(* IEC 61131-3 sources: Industry-PLC-LLM/data/PLCBEAD_repo/PLCBEAD_PLCEmbed-main/PLC-BEAD/Source/GEB/TEMP_SI, 1 file *)

(* ---- TEMP_SI.ST ---- *)
FUNCTION TEMP_SI:REAL
	VAR_INPUT
		RES :	REAL;
		VAR_RS:	REAL;
		TS :	REAL;
	END_VAR

	TEMP_SI := (-7.64E-3 + SQRT(RES/VAR_RS* 6.64E-5 - 0.803E-5)) * 30120.48193 + TS;

END_FUNCTION

PROGRAM program0
  	VAR
		RES :	REAL;
		VAR_RS:	REAL;
		TS :	REAL;
    	CEIL5_OUT : REAL;
  	END_VAR

  	CEIL5_OUT := TEMP_SI(RES, VAR_RS, TS);
END_PROGRAM
